{attribute 'GeneratedUsingTerminal: EL6201-0000-0018'}
{attribute addProperty BoxType "EL6201-0000-0018"}
{attribute addProperty Id "ASI_Inputs_DeviceAT %I*ASI_Inputs_Device_7F2828A5248ASI_StatusAT %I*ASI_Status_279C390313ASI_Outputs_DeviceAT %Q*ASI_Outputs_Device_16036E19248ASI_ControlAT %Q*ASI_Control_2BED18937WcStateAT %I*WcState_9091E0EB2InfoDataAT %I*InfoData_94A18F5E2"}
{attribute addProperty CRC "2305555378"}
{attribute addProperty Size "520"}
TYPE EL6201_896BFBB2 EXTENDS EtcSlaveTerminalBase_947E5A46 :
STRUCT
	{attribute addProperty Name "ASI_Inputs_Device"}
	ASI_Inputs_Device : ASI_Inputs_Device_7F2828A5;
	{attribute addProperty Name "ASI_Status"}
	ASI_Status : ASI_Status_279C3903;
	{attribute addProperty Name "ASI_Outputs_Device"}
	ASI_Outputs_Device : ASI_Outputs_Device_16036E19;
	{attribute addProperty Name "ASI_Control"}
	ASI_Control : ASI_Control_2BED1893;
	{attribute addProperty Name "WcState"}
	WcState : WcState_9091E0EB;
	{attribute addProperty Name "InfoData"}
	InfoData : InfoData_94A18F5E;
END_STRUCT
END_TYPE

(* stored: Version 1.2.0.0, ProductVersion 3.1.4024.9
   DUT EL6201_896BFBB2: Id {b5c547f2-1e0b-4fbb-992e-bc92f39249d5} *)
